INTERFACE I_ListSTRING

METHOD M_Add : BOOL
VAR_INPUT
	Value:		STRING(255);
END_VAR
END_METHOD

METHOD M_Clear : BOOL
END_METHOD

METHOD M_Index : DINT
VAR_INPUT
	Value:	STRING(255);
END_VAR
END_METHOD

METHOD PUBLIC M_Insert : BOOL
VAR_INPUT
	Position:		UDINT;
	Value:			STRING(255);
END_VAR
END_METHOD

METHOD M_Item : STRING(255)
VAR_INPUT
	Index: 	DINT;
END_VAR
END_METHOD

METHOD M_Remove : bool
VAR_INPUT
	Position:			DINT;
END_VAR
END_METHOD

METHOD M_Search : DINT
VAR_INPUT
	Value:		STRING(255);
END_VAR
END_METHOD

PROPERTY P_Length : DINT
GET
END_GET
END_PROPERTY

END_INTERFACE

(* stored: Version 1.1.0.1
   Itf I_ListSTRING: Id {937c5750-ac4a-0c75-3ddd-b288d095682e}
   Method M_Add: Id {7d041429-e10d-09cb-3fcd-bd535d305c8b}
   Method M_Clear: Id {2568afe7-f1ba-0d49-04c6-4cf7f25a949a}
   Method M_Index: Id {4c369575-4541-0c11-19ef-292e554e4ba7}
   Method M_Insert: Id {8c7c3197-9d8e-024f-2384-b75a17732138}
   Method M_Item: Id {905d8954-1c11-0cee-01d2-ea1e30f0ae14}
   Method M_Remove: Id {3d146390-4ec0-0a33-08ae-7d967444c553}
   Method M_Search: Id {5b3ec785-684b-03f5-2c9c-f1a00aa7c91f}
   Property P_Length: Id {dd1a731e-7c76-0405-3a5b-64fd53e98745}
   Get Get: Id {59abc2b2-589e-0023-0109-6a75ba5d563a} *)
